PROGRAM S13_Labeling
VAR
	//工站
	station					: REFERENCE TO FB_Station:=fbstation[13];
	//气缸
	fbHOZCyl_1			:REFERENCE TO FB_Cylinder:=fbCylinder[36];	//	分料气缸1
	//延时
	arTonDelay :ARRAY[1..20] OF TON;
	//返回值
	UdiReturnValue :ARRAY[1..20] OF UDINT;
	//贴标机
	xLabelJobRdySignal:BOOL;//	贴标机JOBRDY信号
	xLabelReadySignal:BOOL;//	贴标机READY信号
	xLabelErrorSignal:BOOL;//	贴标机ERROR信号
	i: INT;
	xQLabelStart: BOOL;			//	贴标机Start 
	xQLabelRibwarn: BOOL; //	贴标机RIBWARN
	xQLabelReset: BOOL;   //	贴标机RESET  
	// 贴标到位传感器
	arSensorReached: ARRAY[1..2]of BOOL;
	
	// 设备停止延时
	tStopDelay: TON;
END_VAR

A_Input();
Alarm();
Delay();
FlowAuto();
FlowInit();
General();
ILC();
TipAuto();
TipManual();
Z_Output();

ACTION A_Input:
//气缸
fbHOZCyl_1.xWP_Sensor:=	IxS11HOZCylWP	;//	贴标处推料气缸¶动点
fbHOZCyl_1.xHP_Sensor:=	IxS11HOZCylHP	;//	贴标处推料气缸¶原点
//贴标机

xLabelJobRdySignal:=IxLabelJobRdySignal	;//	贴标机JOBRDY信号
xLabelReadySignal:=IxLabelReadySignal	;//	贴标机READY信号
xLabelErrorSignal:= NOT IxLabelErrorSignal	;//	贴标机ERROR信号

//贴标机到位传感器
arSensorReached[1]:=IxS11SensorReached1	;//	贴标工位¶检查到位传感器1
arSensorReached[2]:=IxS11SensorReached2;//	贴标工位¶检查到位传感器2
END_ACTION

ACTION Alarm:

station.adwAlarm[1].00:=station.xInitTimeout;	  			//S08Label 初始化超时
END_ACTION

ACTION Delay:
(*arTonDelay[01](IN:= , PT:=T#0.1S , Q=> , ET=> );*)//TipAuto使用
arTonDelay[02](IN:= station.iStepAuto=100 , PT:=T#1S , Q=> , ET=> );//贴标识用
arTonDelay[03](IN:=station.iStepAuto =40  , PT:=stData.TimeS[1] , Q=> , ET=> );//计算贴标延时
arTonDelay[04](IN:= , PT:=T#0.1S , Q=> , ET=> );
arTonDelay[05](IN:= , PT:=T#0.1S , Q=> , ET=> );
arTonDelay[06](IN:= , PT:=T#0.1S , Q=> , ET=> );
arTonDelay[07](IN:= , PT:=T#0.1S , Q=> , ET=> );
arTonDelay[08](IN:= , PT:=T#0.1S , Q=> , ET=> );
arTonDelay[09](IN:= , PT:=T#0.1S , Q=> , ET=> );
END_ACTION

ACTION FlowAuto:

//-----------------------------------------初始化是否完成判断----------------------------------------------
IF NOT station.xInitDone 
THEN
 	station.iStepAuto:=0;
 	station.xDone:=FALSE;
ELSIF station.xRunning  OR   station.xRunningOffProhibit
THEN
//-----------------------------------------动作步骤--------------------------------------------------------
CASE station.iStepAuto OF	  
	0: //----Home Step，等待启动----
		IF station.xDisabled 
			AND station.xCanRun 
			AND NOT fbMachine[1].xStopped 
			AND NOT station.xSingleRunning 
		THEN
			station.xDone:=TRUE;
		END_IF
		
		IF  station.xSingleRunning 
			OR station.xCanRun 
			AND NOT station.xDone 
			AND NOT station.xDisabled 
			AND NOT fbMachine[1].xStopped
		THEN
			station.xCycleEnable:=TRUE;
			station.xDone:= FALSE;  
			station.xRunningOffProhibit := TRUE ;//运行中信号Off禁止
			station.iStepAuto:= 10;
		END_IF
    10: //复位数据 
			xQLabelStart:=FALSE;			//	贴标机Start
			station.iStepAuto:=20;
		20://等待第一个传感器感应到
			IF  arSensorReached[1] THEN
						station.iStepAuto:=30;	
			END_IF
		30://等待两个传感器都感应到
				IF  arSensorReached[1]  AND arSensorReached[2] THEN
						station.iStepAuto:=40;	
			END_IF
		40://计算延时触发贴标
				IF   arTonDelay[03].Q THEN
					station.iStepAuto:=100;
				END_IF
		100://开始触发贴标
					xQLabelStart:=TRUE;			//	贴标机Start
					IF	arTonDelay[02].Q THEN
							station.iStepAuto:=110;
					END_IF							
		110://等待贴标完成
					xQLabelStart:=FALSE;			//	贴标机stop
					station.iStepAuto:=999;

		999://----Single Run Finish----
				station.iStepAuto :=0;
				IF NOT station.xSingleContinuousRun THEN
					station.xSingleRunFlag:=FALSE;
				END_IF
				
				station.xCycleEnable:=FALSE;	
				//station.xDone:=TRUE;
				station.xRunningOffProhibit := FALSE ;//运行中信号Off禁止
	ELSE
		;	
END_CASE



END_IF
END_ACTION

ACTION FlowInit:
IF NOT station.xIniting THEN
  station.iStepInit:=0;    
ELSE
//--------------------------------------------初始化步序----------------------------------
CASE station.iStepInit OF	
 0://  
  	IF station.xIniting THEN	
  	  station.iStepInit:=10;	
  	END_IF	
10://复位数据
    station.iStepInit:=999;	
		xQLabelStart:=FALSE;			//	贴标机Start
999://初始化完成	
	station.iStepInit:=0;
	station.xInitDone:=TRUE;  
END_CASE
END_IF
END_ACTION

ACTION General:
{region "停止"}
tStopDelay(IN:= fbMachine[1].xManualMode, PT:=T#60S , Q=> , ET=> );
IF tStopDelay.Q THEN
		station.xRunningOffProhibit:=FALSE;
ELSIF  station.iStepAuto =10 THEN
		station.xRunningOffProhibit:=TRUE;
END_IF	 
{endregion}
END_ACTION

ACTION ILC:

//---------------------------------------------------工站可执行-------------------------------------------------------
station.xCanRun :=TRUE ;

//---------------------------------------------------气缸动作条件-------------------------------------------
fbHOZCyl_1.xOffILC	:=	TRUE	;
fbHOZCyl_1.xOnILC	:=	TRUE; 


//---------------------------------------------------伺服动作条件-------------------------------------------
END_ACTION

ACTION TipAuto:

//------------------------------------------------AutoTip Cylinder--------------------------------

//------------------------------------------------AutoTip Servo--------------------------------
//**************************************
END_ACTION

ACTION TipManual:
//--------------------------------------------ManualTip------------------------------------------------------

//-------------------------------------------气缸提示---------------------------------------------------------




/////////////////////////////////////////////////////////////////////////////////////////////////////////////////
END_ACTION

ACTION Z_Output:
(**************************气缸输出********************************)
QxS11HOZCylWP	:=fbHOZCyl_1.xWP_Valve;//	贴标处推料气缸¶动点
QxS11HOZCylHP	:=fbHOZCyl_1.xHP_Valve;//	贴标处推料气缸¶原点
//贴标机
QxLabelStart	:=xQLabelStart;			//	贴标机Start
QxLabelRibwarn:=xQLabelRibwarn;	//	贴标机RIBWARN
QxLabelReset	:=xQLabelReset;		//	贴标机RESET
END_ACTION

END_PROGRAM

(* stored: Version 1.1.0.1, ProductVersion 3.1.4024.9
   POU S13_Labeling: Id {e6e1a2a9-780c-4003-bca7-0316b25c817d}, SpecialFunc None
   Action A_Input: Id {08bf5b2d-c23a-4b9f-bc0b-d78d0ef357a0}
   Action Alarm: Id {a33f9682-7f1b-43f4-848a-88bf388c8dd9}
   Action Delay: Id {640cd6ea-e634-4695-b63f-ca35a17c42ab}
   Action FlowAuto: Id {9d4d8677-e15d-419a-b731-9583a551307c}
   Action FlowInit: Id {40d5274c-5ab2-4ba2-a9ce-2aa53d171fca}
   Action General: Id {7e130351-797e-4ca7-9bb7-b3cd5e7898e1}
   Action ILC: Id {a47065cb-3ca4-400c-a537-51952fd23503}
   Action TipAuto: Id {e4cfd73c-4866-4896-867d-52e2f450d72f}
   Action TipManual: Id {096ba1af-e1e4-4b9f-9361-432b4bd5211e}
   Action Z_Output: Id {58bab82e-5ef1-477c-83be-2769659c9d33} *)
